// TIA Portal V21 export
TYPE "Caps_Config"
   STRUCT
      "@_HMI" : Struct
         s_Name { S7_SetPoint := 'True'} : String;
      END_STRUCT;
      "@_CFG" : Struct
         x_CapsFeeder { S7_SetPoint := 'True'} : Bool;   // Abilitazione - Orientatore tappi
         x_CapsFeederReverse { S7_SetPoint := 'True'} : Bool;   // Abilitazione - Marcia indietro orientatore tappi
         x_CheckCapsFeederRotation { S7_SetPoint := 'True'} : Bool;   // Abilitazione - Controllo Rotazione orientatore tappi
         x_CapsFeederAlwaysRunning { S7_SetPoint := 'True'} : Bool;   // Abilitazione - Marcia orientatore senza chiamata da canale tappi
         x_CapsFeederChangeSpeed { S7_SetPoint := 'True'} : Bool;   // Abilitazione - Cambio Velocità orientatore tappi
         x_VacuumPump { S7_SetPoint := 'True'} : Bool;   // Abilitazione - Pompa del Vuoto
         x_CheckCapInverted { S7_SetPoint := 'True'} : Bool;   // Abilitazione - Controllo Tappo Rovesciato nel Canale
         x_LightUV { S7_SetPoint := 'True'} : Bool;   // Abilitazione - Lampada Sterilizzazione UV
         x_EmptyChannel { S7_SetPoint := 'True'} : Bool;   // Abilitazione - Svuotamento Canale
         x_CapsElevator { S7_SetPoint := 'True'} : Bool;   // Abilitazione - Elevatore tappi
         x_CapsBelt { S7_SetPoint := 'True'} : Bool;   // Abilitazione - Nastro tappi
         x_NBNC { S7_SetPoint := 'True'} : Bool;   // Abilitazione - Sgancio Tappo
         x_HeadRot { S7_SetPoint := 'True'} : Bool;   // Abilitazione - Rotazione Teste
         x_AntirotationBelt { S7_SetPoint := 'True'} : Bool;   // Abilitazione - Cinghia anti rotazione
         i_NrChannel { S7_SetPoint := 'True'} : Int;   // Numero canale in uso
         f_KFactor { S7_SetPoint := 'True'} : Real;   // Coefficente per calcolo velocità rotazione teste
         PT { S7_SetPoint := 'True'} : Array[0..19] of Time;
      END_STRUCT;
   END_STRUCT;
   // // "@_CFG".PT[0] : Ton marcia pompa del vuoto
   // // "@_CFG".PT[1] : Ton allarme mancanza tappi nel canale
   // // "@_CFG".PT[2] : Toff allarme mancanza tappi nel canale
   // // "@_CFG".PT[3] : Ton consenso di marcia a orientatore tappi
   // // "@_CFG".PT[4] : Toff consenso di marcia a orientatore tappi
   // // "@_CFG".PT[5] : Ton SQ ctrl tappo rovesciato nel canale
   // // "@_CFG".PT[6] : Toff apertura sportello lampada UV
   // // "@_CFG".PT[7] : Ton SQ on ctrl rotazione orientatore tappi
   // // "@_CFG".PT[8] : Ton consenso di marcia a elevatore tappi
   // // "@_CFG".PT[9] : Toff consenso di marcia a elevatore tappi
   // // "@_CFG".PT[10] : Toff aria tappatore
   // // "@_CFG".PT[11] : Ton aria tappatore attiva
   // // "@_CFG".PT[12] : Ton marcia orientatore tappi
   // // "@_CFG".PT[13] : Ton cambio velocità orientatore tappi
   // // "@_CFG".PT[14] : Ton SQ off ctrl tappo rovesciato nel canale
   // // "@_CFG".PT[15] : Ton consenso di marcia a nastro tappi
   // // "@_CFG".PT[16] : Toff consenso di marcia a nastro tappi
END_TYPE
